INTERFACE ITF_BaseTopElement_HMI_Connector_Command

END_INTERFACE

(* stored: Version 1.1.0.1
   Itf ITF_BaseTopElement_HMI_Connector_Command: Id {7099e25d-4c3a-058f-13e0-64e3c1f21687} *)
